{attribute addProperty BoxType "EJ3004-0000-0020"}
{attribute addProperty Id "StatusAT %I*Status_F0C7FE3C658.1251ValueAT %I*INT16217"}
{attribute addProperty CRC "3786149730"}
{attribute addProperty SizeInBites "81"}
{attribute addProperty SizeInBytes "10.125"}
TYPE AI_Standard_Channel_E1AC0F62 :
STRUCT
	{attribute addProperty Name "Status"}
	Status AT %I* : Status_F0C7FE3C;
	{attribute addProperty Name "Value"}
	Value AT %I* : INT;
END_STRUCT
END_TYPE

(* stored: Version 1.2.0.0, ProductVersion 3.1.4024.9
   DUT AI_Standard_Channel_E1AC0F62: Id {2a6bf1eb-635c-457f-9e6e-824d77752417} *)
